Staubli VAL3: PALLET.dtx

public TrajPallet tTraj{}
